{attribute 'OPC.UA.DA.StructuredType':=1}
TYPE ST_QrSkillSpecific :
STRUCT
    CameraReady     : BOOL := FALSE;

    Result          : STRING(255) := '';
    Quality         : REAL := 0.0;

    CodeType        : STRING(32) := '';
END_STRUCT
END_TYPE

(* stored: Version 1.1.0.1, ProductVersion 3.1.4026.18
   DUT ST_QrSkillSpecific: Id {31e14e33-bcd8-4eb4-8cdb-67a96a5d4a8a} *)
